// TIA Portal V18 export
FUNCTION_BLOCK "SideShifter"   // FB2, LAD
{ S7_Optimized_Access := 'TRUE' }
// stored: MemoryReserve 100, SetENOAutomatically false
   VAR_INPUT
      Hydraulic_Up : Bool;
      Hydraulic_Down : Bool;
      Hydraulic_Unit : Bool;
      Homing1 : Bool;
      Homing2 : Bool;
      Homing3 : Bool;
      Safety : Bool;
   END_VAR
   VAR_OUTPUT
      Hydraulic_Actuator1_Up : Bool;
      Hydraulic_Actuator1_Down : Bool;
      Hydraulic_Actuator2_Up : Bool;
      Hydraulic_Actuator2_Down : Bool;
      Hydraulic_Unit1 : Bool;
      Hydraulic_Unit2 : Bool;
   END_VAR
BEGIN
END_FUNCTION_BLOCK
